{attribute 'qualified_only'}
{attribute 'strict'}
TYPE DevStates :
(
	NOOP := 0,
	IDLE,
 	RECEIVING,
	PROC,
	SENDING,
	ERR
);
END_TYPE

(* stored: Version 1.1.0.1, ProductVersion 3.1.4024.15
   DUT DevStates: Id {df7e0902-f6aa-4a26-afad-39b511212b96} *)
